PROGRAM MainScreenBindings
VAR
	PercentageLabel_Invisible : BOOL;
	ReactorLowerTemperatureTextField_TextVariable : INT;
	UpperTemperatureTextField_TextVariable : INT;
	ReactorTemperatureSetpointTextField_TextVariable : INT;
	RectorTemperatureControlModeButton_ToggleVariable : BOOL;
	
	ReactorUpperTemperatureTextField_TextVariable : INT;
	RectorTemperatureControlModeButton_TextVariable : STRING; 
	
	SlurryOutValveLamp_Variable : BOOL;
	
	ReactorTemperatureControlPercentageTextField_TextVariable : INT;
	ReactorTemperatureControlPercentageTextField_Invisible : BOOL;
	ReactorTemperatureContactorButton_ToggleColor : BOOL;
	ReactorTemperatureContactorButton_Invisible : BOOL;
	ReactorTemperatureContactorButton_ToggleVariable : BOOL;
	PidParamMenuButton_ToggleVariable : BOOL;
	PidParamMenuButton_Invisible : BOOL;
	PidParamMenuFrame_Invisible : BOOL;
	ReactorTemperatureContactorClosedLine_Invisible : BOOL;
	ReactorTemperatureContactorOpenLine_Invisible : BOOL;
	ReactorTemperatureContactorLamp_Variable : BOOL;
	ReactorBackgroundRectangle_ToggleColor : BOOL;
	ReactorUpperUpperLevelReactangle_Invisible : BOOL;
	ReactorUpperLevelRectangle_Invisible : BOOL;
	ReactorLowerLevelReactangle_Invisible : BOOL;
	ReactorUpperLevelLamp_Variable : BOOL;
	ReactorLowerLevelLamp : BOOL;
	SlurryInValveOpenTimeTextField_TextVariable : INT;
	SlurryInValveClosedTimeTextField_TextVariable : INT;
	SlurryInValveFrame_valve_toggleColor : BOOL;
	SlurryInValveFrame_valve_tapVariable : BOOL;
	SlurryInValveLamp_Variable : BOOL;
	SlurryInValveControlModeButton_ToggleColor : BOOL;
	SlurryInValveControlModeButton_ToggleVariable : BOOL;
	SlurryInValveControlModeButton_TextVariable : STRING;
	SlurryInLine1_ToggleColor : BOOL;
	SlurryInLine2_ToggleColor : BOOL;

	SlurryInValveControlModeButton_Invisible : BOOL;
	ReactorPressureTextField_TextVariable : INT;
	UpperIntervalSlurryOnUpperTextField_TextVariable : INT;
	UpperIntervalSlurryOnNotUpperTextField_TextVariable : INT;
	UpperIntervalSlurryOffUpperTextField_TextVariable : INT;
	LowerIntervalSlurryOnUpperTextField_TextVariable : INT;
	LowerIntervalSlurryOnNotUpperTextField_TextVariable : INT;
	LowerIntervalSlurryOffUpperTextField_TextVariable : INT;
	SlurryOutValveFrame_valve_toggleColor : BOOL;
	SlurryOutValveFrame_valve_tapVariable : BOOL;
	SlurryInArrow_ToggleColor : BOOL;
	SlurryOutLine1_ToggleColor : BOOL;
	SlurryOutLine2_ToggleColor : BOOL;
	SlurryOutLine3_ToggleColor : BOOL;
	SlurryOutTriangle_ToggleColor : BOOL;
	SlurryOutValveButton_Invisible : BOOL;
	SlurryOutValveButton_TextVariable : STRING;
	SlurryOutValveButton_ToggleColor : BOOL;
	SlurryOutValveButton_ToggleVariable : BOOL;
	
	SlurryOutControlModeButton_TextVariable : STRING;
	SlurryOutControlModeButton_ToggleColor  : BOOL;
	SlurryOutControlModeButton_ToggleVariable : BOOL;
	
	StartMatlabButton_TextVariable : STRING;
	StartMatlabButton_Color : DWORD;
	StartMatlabButton_DeactivateInputs  : BOOL;
	ProgramNamePrefixTextField_TextVariable : STRING;
	PreHeaterTemperatureTextField_TextVariable : DINT;
	PreHeaterTemperatureSetpointTextField_TextVariable : DINT;
	Co2FlowTextField_TextVariable : DINT;
	Co2PressureTextField_TextVariable : DINT;
	Co2PressureSetpointTextField_TextVariable : DINT;
	SeperatorTemperatureTextField_TextVariable : DINT;
	SeparatorTemperatureSetpointTextField_TextVariable : DINT;
	
END_VAR


IF RectorTemperatureControlModeButton_ToggleVariable THEN
	RectorTemperatureControlModeButton_TextVariable := 'AUTO';
ELSE
	RectorTemperatureControlModeButton_TextVariable := 'MAN';
END_IF

(*** Outlet valve HMI state ***)
IF GVL_IO.reactorOutletValve = 1 THEN
	//LevelControl.sLevelValveState := 'CLOSE';
	MainScreenBindings.SlurryOutValveButton_TextVariable := 'CLOSE';
//	sLevelValveState := 'CLOSE';
END_IF
IF GVL_IO.reactorOutletValve = 0 THEN
	//LevelControl.sLevelValveState := 'OPEN';
	MainScreenBindings.SlurryOutValveButton_TextVariable := 'OPEN';
//	sLevelValveState := 'OPEN';
END_IF

(*** Inlet valve HMI state ***)
IF NOT GVL_IO.reactorInletValve THEN
	//PressureControl.sFillingValveState := 'OPEN';
	MainScreenBindings.SlurryInValveControlModeButton_TextVariable := 'OPEN';
//	sFillingValveState := 'OPEN';
ELSE
	//PressureControl.sFillingValveState := 'CLOSE';
	MainScreenBindings.SlurryInValveControlModeButton_TextVariable := 'CLOSE';
//	sFillingValveState := 'CLOSE';
END_IF




PercentageLabel_Invisible := RectorTemperatureControlModeButton_ToggleVariable;//ReactorTemperatureControl.bTemperatureControlSwitch;
ReactorLowerTemperatureTextField_TextVariable := ReactorTemperature.lowerTemperature;//ReactorTemperatureControl.iTemperatureDisplayValue;
ReactorUpperTemperatureTextField_TextVariable := ReactorTemperature.upperTemperature;//ReactorTemperatureControl.iTemperatureLowerDisplayValue;
ReactorTemperature.temperatureSetpoint := ReactorTemperatureSetpointTextField_TextVariable;//ReactorTemperatureSetpointTextField_TextVariable := ReactorTemperature.temperatureSetpoint;//ReactorTemperatureControl.iTemperatureSetpoint;
//RectorTemperatureControlModeButton_TextVariable := ReactorTemperatureControl.sTemperatureControlState;
ReactorTemperature.autoControlSelected := RectorTemperatureControlModeButton_ToggleVariable;//ReactorTemperatureControl.bTemperatureControlSwitch := RectorTemperatureControlModeButton_ToggleVariable;// OUTPUT
ReactorTemperature.manualControlPercentage := ReactorTemperatureControlPercentageTextField_TextVariable;//ReactorTemperatureControlPercentageTextField_TextVariable := ReactorTemperature.manualControlPercentage;//ReactorTemperatureControl.iTemperatureControlPercentage;
ReactorTemperatureControlPercentageTextField_Invisible := RectorTemperatureControlModeButton_ToggleVariable; //ReactorTemperatureControl.bTemperatureControlSwitch;
ReactorTemperatureContactorButton_Invisible := ReactorTemperatureControlPercentageTextField_TextVariable > 0 OR RectorTemperatureControlModeButton_ToggleVariable; //ReactorTemperatureControl.iTemperatureControlPercentage > 0 OR ReactorTemperatureControl.bTemperatureControlSwitch= 1;
ReactorTemperature.temperatureContactorCommand := ReactorTemperatureContactorButton_ToggleVariable;//GVL_IO.reactorTemperatureContactor := ReactorTemperatureContactorButton_ToggleVariable;// OUTPUT
//ReactorTemperatureControl.bPIDcontrolParameterMenu := PidParamMenuButton_ToggleVariable;// OUTPUT
PidParamMenuButton_Invisible := RectorTemperatureControlModeButton_ToggleVariable;//ReactorTemperatureControl.bTemperatureControlSwitch;
PidParamMenuFrame_Invisible := NOT PidParamMenuButton_ToggleVariable OR RectorTemperatureControlModeButton_ToggleVariable;//NOT PidParamMenuButton_ToggleVariable OR ReactorTemperatureControl.bTemperatureControlSwitch;//NOT ReactorTemperatureControl.bPIDcontrolParameterMenu OR ReactorTemperatureControl.bTemperatureControlSwitch;
ReactorTemperatureContactorClosedLine_Invisible := NOT GVL_IO.reactorTemperatureContactor;
ReactorTemperatureContactorOpenLine_Invisible := GVL_IO.reactorTemperatureContactor;
ReactorTemperatureContactorLamp_Variable := GVL_IO.reactorTemperatureContactor;
ReactorBackgroundRectangle_ToggleColor := (RectorTemperatureControlModeButton_ToggleVariable) 
										OR (ReactorTemperatureControlPercentageTextField_TextVariable > 0) 
										OR ((ReactorTemperatureControlPercentageTextField_TextVariable = 0) AND (GVL_IO.reactorTemperatureContactor = 1));//(ReactorTemperatureControl.bTemperatureControlSwitch) OR (ReactorTemperatureControl.iTemperatureControlPercentage > 0) OR ((ReactorTemperatureControl.iTemperatureControlPercentage = 0) AND (GVL_IO.reactorTemperatureContactor = 1));
ReactorUpperUpperLevelReactangle_Invisible := (NOT GVL_IO.reactorLevelHigherHigh);
ReactorUpperLevelRectangle_Invisible := (NOT GVL_IO.reactorLevelLow) OR (GVL_IO.reactorLevelHigherHigh);
ReactorLowerLevelReactangle_Invisible := (NOT GVL_IO.reactorLevelHigh) OR (GVL_IO.reactorLevelLow);
ReactorUpperLevelLamp_Variable := GVL_IO.reactorLevelHigh;
ReactorLowerLevelLamp := GVL_IO.reactorLevelLow;
SlurryInValveOpenTimeTextField_TextVariable := ReactorLevelAndPressure.fillingValveOpenInterval;
SlurryInValveClosedTimeTextField_TextVariable := ReactorLevelAndPressure.fillingValveCloseInterval;
SlurryInValveFrame_valve_toggleColor := GVL_IO.reactorInletValve;
GVL_IO.reactorInletValve := SlurryInValveFrame_valve_tapVariable; // OUTPUT
SlurryInValveLamp_Variable := GVL_IO.reactorInletValve;
SlurryInValveControlModeButton_ToggleColor := GVL_IO.reactorInletValve;
//SlurryInValveControlModeButton_TextVariable := ReactorLevelAndPressure.sFillingValveState;
GVL_IO.reactorInletValve := SlurryInValveControlModeButton_ToggleVariable;
SlurryInLine1_ToggleColor := GVL_IO.reactorInletValve;
SlurryInLine2_ToggleColor := GVL_IO.reactorInletValve;

SlurryInValveControlModeButton_Invisible := ReactorLevelAndPressure.sLevelControlState = 'AUTO';
ReactorPressureTextField_TextVariable := ReactorLevelAndPressure.iPressureScaledValue;
UpperIntervalSlurryOnUpperTextField_TextVariable := ReactorLevelAndPressure.PressureUpperInterVal_1;
UpperIntervalSlurryOnNotUpperTextField_TextVariable := ReactorLevelAndPressure.PressureUpperInterVal_2;
UpperIntervalSlurryOffUpperTextField_TextVariable := ReactorLevelAndPressure.PressureUpperInterVal_3;
LowerIntervalSlurryOnUpperTextField_TextVariable := ReactorLevelAndPressure.PressureLowerInterval_1;
LowerIntervalSlurryOnNotUpperTextField_TextVariable := ReactorLevelAndPressure.PressureLowerInterval_2;
LowerIntervalSlurryOffUpperTextField_TextVariable := ReactorLevelAndPressure.PressureLowerInterval_3;
SlurryOutValveFrame_valve_toggleColor := GVL_IO.reactorOutletValve;
GVL_IO.reactorOutletValve := SlurryOutValveFrame_valve_tapVariable;// OUTPUT
SlurryInArrow_ToggleColor := GVL_IO.reactorInletValve;
SlurryOutLine1_ToggleColor := GVL_IO.reactorOutletValve;
SlurryOutLine2_ToggleColor := GVL_IO.reactorOutletValve;
SlurryOutLine3_ToggleColor := GVL_IO.reactorOutletValve;
SlurryOutTriangle_ToggleColor := GVL_IO.reactorOutletValve;
SlurryOutValveLamp_Variable := GVL_IO.reactorOutletValve;
SlurryOutValveButton_Invisible := ReactorLevelAndPressure.sLevelControlState = 'AUTO';
//SlurryOutValveButton_TextVariable := ReactorLevelAndPressure.sLevelValveState;
SlurryOutValveButton_ToggleColor := GVL_IO.reactorOutletValve;
GVL_IO.reactorOutletValve := SlurryOutValveButton_ToggleVariable;// OUTPUT

SlurryOutControlModeButton_TextVariable := ReactorLevelAndPressure.sLevelControlState;
SlurryOutControlModeButton_ToggleColor := SlurryOutControlModeButton_ToggleVariable;//ReactorLevelAndPressure.bLevelControlSwitch;
ReactorLevelAndPressure.bLevelControlSwitch := SlurryOutControlModeButton_ToggleVariable; // TARKISTA? // OUTPUT

StartMatlabButton_TextVariable := RunMATLAB.sMatlabRunningState;
StartMatlabButton_Color := RunMATLAB.dMatlabBtnColor;
StartMatlabButton_DeactivateInputs := RunMATLAB.dMatlabBtnColor = 16#FFFFFF00;
ProgramNamePrefixTextField_TextVariable := GVL_OPC.OPC_ProgramNamePrefix;
PreHeaterTemperatureTextField_TextVariable := SerialCommunicationHandler.preHeaterTemperatureMeasurement;
PreHeaterTemperatureSetpointTextField_TextVariable := SerialCommunicationHandler.preHeaterTemperatureSetpoint;
Co2FlowTextField_TextVariable := SerialCommunicationHandler.flowMeasurement;
Co2PressureTextField_TextVariable := SerialCommunicationHandler.pumpingPressureMeasurement;
Co2PressureSetpointTextField_TextVariable := SerialCommunicationHandler.pumpingPressureSetpoint;
SeperatorTemperatureTextField_TextVariable := SerialCommunicationHandler.separatorTemperatureMeasurement;
SeparatorTemperatureSetpointTextField_TextVariable := SerialCommunicationHandler.separatorTemperatureSetpoint;

PidParamMenuFrame_Invisible := NOT PidParamMenuButton_ToggleVariable OR RectorTemperatureControlModeButton_ToggleVariable;//NOT PidParamMenuButton_ToggleVariable OR ReactorTemperatureControl.bTemperatureControlSwitch;//NOT ReactorTemperatureControl.bPIDcontrolParameterMenu OR ReactorTemperatureControl.bTemperatureControlSwitch;

END_PROGRAM

(* stored: Version 1.1.0.1, ProductVersion 3.1.4024.9
   POU MainScreenBindings: Id {4a3b100e-d510-409e-8f4e-7c5919608164}, SpecialFunc None *)
